{attribute 'GeneratedUsingTerminal: EK1814-0000-0016'}
{attribute addProperty BoxType "EK1814-0000-0016"}
{attribute addProperty Id "OutputAT %Q*BOOL1"}
{attribute addProperty CRC "1120571895"}
{attribute addProperty Size "1"}
TYPE Channel_42CA91F7 :
STRUCT
	{attribute addProperty Name "Output"}
	Output AT %Q* : BOOL;
END_STRUCT
END_TYPE

(* stored: Version 1.2.0.0, ProductVersion 3.1.4024.9
   DUT Channel_42CA91F7: Id {b4326b4d-eed4-40b0-84ea-4ec14f54db7c} *)
